{attribute 'qualified_only'}
VAR_GLOBAL
END_VAR

(* stored: Version 1.1.0.1
   GVL Testy: Id {f2c4afe0-0b43-448f-8de8-b7695b06ba09} *)
